// TIA Portal V15.1 export
// export: Created 2020-12-07T09:03:51.8959299Z, ExportSetting WithDefaults, WithReadOnly, DisplayName Totally Integrated Automation Portal, DisplayVersion V15.1 Update 4, DisplayName TIA Portal Openness, DisplayVersion V15.1, DisplayName SINAMICS Startdrive Advanced, DisplayVersion V15.1 Update3, DisplayName SINAMICS Startdrive G110M, G120, G120C, G120D, G120P, DisplayVersion V15.1 Update3, DisplayName SINAMICS Startdrive G130, G150, S120, S150, SINAMICS MV, S210, DisplayVersion V15.1 Update3, DisplayName STEP 7 Professional, DisplayVersion V15.1 Update 4, DisplayName STEP 7 Safety, DisplayVersion V15.1, DisplayName WinCC Professional, DisplayVersion V15.1 Update 4
VAR_GLOBAL   // PLC tag table "INPUT_ST_A"
   "SQ84/BA" AT %I2000.0 : Bool;
   "SQ85/BA" AT %I2001.0 : Bool;
   "SQ86/BA" AT %I2000.1 : Bool;
   "SQ87/BA" AT %I2001.1 : Bool;
   "SQ57/BA" AT %I2000.2 : Bool;
   "SQ58/BA" AT %I2001.2 : Bool;
   "SQ59/BA" AT %I2000.3 : Bool;
   "SQ60/BA" AT %I2001.3 : Bool;
   "SQ73/BA" AT %I2000.4 : Bool;
   "SQ74/BA" AT %I2001.4 : Bool;
   "SQ31/BA" AT %I2000.5 : Bool;
   "SQ32/BA" AT %I2001.5 : Bool;
   "FTC1/BA" AT %I2000.7 : Bool;
   "SQ15/BA" AT %I2001.6 : Bool;
   "FTC2/BA" AT %I2000.6 : Bool;
   "FTC3/BA" AT %I2001.7 : Bool;
   "SQ61/BA" AT %I2002.0 : Bool;
   "SQ62/BA" AT %I2003.0 : Bool;
   "SQ66/BA" AT %I2002.1 : Bool;
   "SQ67/BA" AT %I2003.1 : Bool;
   "SQ68/BA" AT %I2002.2 : Bool;
   "SQ72/BA" AT %I2003.2 : Bool;
   "SQ8/BA" AT %I2002.3 : Bool;   // // NC
   "SQ9/BA" AT %I2003.3 : Bool;   // // NC
   "SQ80/BA" AT %I2002.4 : Bool;
   "SQ81/BA" AT %I2003.4 : Bool;
   "FTC15/BA" AT %I2002.5 : Bool;   // Scivolo troppo pieno
   "FTC92/BA" AT %I2003.5 : Bool;   // Presenza rullo su OP30
   "FTC93/BA" AT %I2002.6 : Bool;   // Presenza rullo su OP20
   "FTC94/BA" AT %I2003.6 : Bool;   // Presenza rullo su OP10
   "SQ_SPARE_31/BA" AT %I2002.7 : Bool;
   "SQ_SPARE_32/BA" AT %I2003.7 : Bool;
   "SQ_SPARE_33/BA" AT %I2004.0 : Bool;   // // NC
   "SQ_SPARE_34/BA" AT %I2005.0 : Bool;   // // NC
   "SQ_SPARE_35/BA" AT %I2004.1 : Bool;   // // NC
   "SQ_SPARE_36/BA" AT %I2005.1 : Bool;   // // NC
   "SQ_SPARE_37/BA" AT %I2004.2 : Bool;   // // NC
   "SQ_SPARE_38/BA" AT %I2005.2 : Bool;   // // NC
   "SQ_SPARE_39/BA" AT %I2004.3 : Bool;
   "SQ_SPARE_40/BA" AT %I2005.3 : Bool;
   "SQ_SPARE_41/BA" AT %I2004.4 : Bool;
   "SQ_SPARE_42/BA" AT %I2005.4 : Bool;
   "SQ_SPARE_43/BA" AT %I2004.5 : Bool;
   "SQ_SPARE_44/BA" AT %I2005.5 : Bool;
   "SQ_SPARE_45/BA" AT %I2004.6 : Bool;
   "SQ_SPARE_46/BA" AT %I2005.6 : Bool;
   "SQ_SPARE_47/BA" AT %I2004.7 : Bool;
   "SQ_SPARE_48/BA" AT %I2005.7 : Bool;
   "SQ44/BA" AT %I2100.0 : Bool;
   "SQ45/BA" AT %I2101.0 : Bool;
   "SQ88/BA" AT %I2100.1 : Bool;
   "SQ89/BA" AT %I2101.1 : Bool;
   "SQ48/BA" AT %I2100.2 : Bool;
   "SQ49/BA" AT %I2101.2 : Bool;
   "SQ50/BA" AT %I2100.3 : Bool;
   "SQ51/BA" AT %I2101.3 : Bool;
   "SQ75/BA" AT %I2100.4 : Bool;
   "SQ76/BA" AT %I2101.4 : Bool;
   "SQ18/BA" AT %I2100.5 : Bool;
   "SQ19/BA" AT %I2101.5 : Bool;
   "SQ97/BA" AT %I2100.6 : Bool;
   "SQ17/BA" AT %I2101.6 : Bool;
   "SQ98/BA" AT %I2100.7 : Bool;
   "SQ_SPARE_64/BA" AT %I2101.7 : Bool;
   "SQ_SPARE_65/BA" AT %I2102.0 : Bool;   // // NC
   "SQ_SPARE_66/BA" AT %I2103.0 : Bool;   // // NC
   "SQ_SPARE_67/BA" AT %I2102.1 : Bool;   // // NC
   "SQ_SPARE_68/BA" AT %I2103.1 : Bool;   // // NC
   "SQ_SPARE_69/BA" AT %I2102.2 : Bool;   // // NC
   "SQ_SPARE_70/BA" AT %I2103.2 : Bool;   // // NC
   "SQ_SPARE_71/BA" AT %I2102.3 : Bool;
   "SQ_SPARE_72/BA" AT %I2103.3 : Bool;
   "SQ_SPARE_73/BA" AT %I2102.4 : Bool;
   "SQ_SPARE_74/BA" AT %I2103.4 : Bool;
   "SQ_SPARE_75/BA" AT %I2102.5 : Bool;
   "SQ_SPARE_76/BA" AT %I2103.5 : Bool;
   "SQ_SPARE_77/BA" AT %I2102.6 : Bool;
   "SQ_SPARE_78/BA" AT %I2103.6 : Bool;
   "SQ_SPARE_79/BA" AT %I2102.7 : Bool;
   "SQ_SPARE_80/BA" AT %I2103.7 : Bool;
   "SQ69/BA" AT %I2104.0 : Bool;
   "SQ70/BA" AT %I2105.0 : Bool;
   "SQ71/BA" AT %I2104.1 : Bool;
   "SQ77/BA" AT %I2105.1 : Bool;
   "SQ78/BA" AT %I2104.2 : Bool;
   "SQ79/BA" AT %I2105.2 : Bool;   // // NC
   "SQ6/BA" AT %I2104.3 : Bool;
   "SQ7/BA" AT %I2105.3 : Bool;
   "SQ82/BA" AT %I2104.4 : Bool;
   "SQ83/BA" AT %I2105.4 : Bool;
   "SQ_SPARE_91/BA" AT %I2104.5 : Bool;
   "SQ_SPARE_92/BA" AT %I2105.5 : Bool;
   "SQ_SPARE_93/BA" AT %I2104.6 : Bool;
   "SQ_SPARE_94/BA" AT %I2105.6 : Bool;
   "SQ_SPARE_95/BA" AT %I2104.7 : Bool;
   "SQ_SPARE_96/BA" AT %I2105.7 : Bool;
   "STO_AZ2/BA" AT %I4.0 : Bool;   // // NC
   "STO_AZ3/BA" AT %I4.1 : Bool;   // // NC
   "STO_AZ11/BA" AT %I4.2 : Bool;   // // NC
   "STO_AZ14/BA" AT %I4.3 : Bool;   // // NC
   "STO_AZ18/BA" AT %I4.4 : Bool;   // // NC
   "STO_AZ20/BA" AT %I4.5 : Bool;   // // NC
   "STO_AZ22/BA" AT %I4.6 : Bool;   // // NC
   "STO_AZ24/BA" AT %I4.7 : Bool;   // // NC
   "STO_AZ4/BA" AT %I5.0 : Bool;   // // NC
   "STO_AZ5/BA" AT %I5.1 : Bool;   // // NC
   "STO_AZ6/BA" AT %I5.2 : Bool;   // // NC
   "STO_AZ7/BA" AT %I5.3 : Bool;   // // NC
   "STO_AZ8/BA" AT %I5.4 : Bool;   // // NC
   "STO_AZ9/BA" AT %I5.5 : Bool;   // // NC
   "STO_AZ10/BA" AT %I5.6 : Bool;   // // NC
   "STO_AZ12/BA" AT %I5.7 : Bool;   // // NC
   "STO_AZ13/BA" AT %I6.0 : Bool;   // // NC
   "STO_AZ15/BA" AT %I6.1 : Bool;   // // NC
   "STO_AZ17/BA" AT %I6.2 : Bool;   // // NC
   "STO_AZ19/BA" AT %I6.3 : Bool;   // // NC
   "STO_AZ21/BA" AT %I6.4 : Bool;   // // NC
   "STO_AZ23/BA" AT %I6.5 : Bool;   // // NC
   "STO_AZ25/BA" AT %I6.6 : Bool;   // // NC
   "STO_AZ26/BA" AT %I6.7 : Bool;   // // NC
   "OIL_PUMP_FAULT/BA" AT %I7.0 : Bool;
   "EMG_OK/BA" AT %I7.1 : Bool;
   "OIL_HIGH_TEMP/BA" AT %I7.2 : Bool;
   "OIL_LOW_LEVEL/BA" AT %I7.3 : Bool;
   "LASER_ERROR/BA" AT %I7.4 : Bool;   // // NC
   "AZ27_RUN/BA" AT %I7.6 : Bool;   // // NC
   "AZ27_FAULT/BA" AT %I7.7 : Bool;   // // NC
   "LOAD_CELL_SX_FAULT/BA" AT %I8.0 : Bool;
   "PS_KOSTYRCA_ENDCAP_SX/BA" AT %I8.1 : Bool;
   "PS_KOSTYRCA_SEEGER_SX/BA" AT %I8.2 : Bool;
   "PS_KOSTYRCA_ENDCAP_DX/BA" AT %I8.3 : Bool;
   "PS_KOSTYRCA_SEEGER_DX/BA" AT %I8.4 : Bool;
   "LOAD_CELL_DX_FAULT/BA" AT %I8.5 : Bool;
   "TLB1/BA" AT %IW2 : Int;   // Load cell endcap sx
   "TLB2/BA" AT %IW0 : Int;   // Load cell endcap dx
   "TOR1/BA" AT %IW10 : Int;   // Torsiometro
   "FTC5/BA" AT %I2006.0 : Bool;
   "FTC7/BA" AT %I2006.1 : Bool;
   "SQ_SPARE_99/BA" AT %I2006.2 : Bool;
   "FTC90/BA" AT %I2006.3 : Bool;   // Presenza Endcap SX
   "SQ_SPARE_101/BA" AT %I2006.4 : Bool;
   "SQ_SPARE_102/BA" AT %I2006.5 : Bool;
   "SQ_SPARE_103/BA" AT %I2006.6 : Bool;
   "SQ_SPARE_104/BA" AT %I2006.7 : Bool;
   "FTC6/BA" AT %I2007.0 : Bool;
   "SQ95/BA" AT %I2007.1 : Bool;
   "SQ_SPARE_107/BA" AT %I2007.2 : Bool;
   "SQ96/BA" AT %I2007.3 : Bool;
   "SQ_SPARE_109/BA" AT %I2007.4 : Bool;
   "SQ_SPARE_110/BA" AT %I2007.5 : Bool;
   "SQ_SPARE_111/BA" AT %I2007.6 : Bool;
   "SQ_SPARE_112/BA" AT %I2007.7 : Bool;
   "SQ_SPARE_113/BA" AT %I2106.0 : Bool;
   "SQ_SPARE_114/BA" AT %I2106.1 : Bool;
   "SQ_SPARE_115/BA" AT %I2106.2 : Bool;
   "SQ_SPARE_116/BA" AT %I2106.3 : Bool;
   "FTC91/BA" AT %I2106.4 : Bool;   // Presenza Endcap DX
   "SQ_SPARE_118/BA" AT %I2106.5 : Bool;
   "SQ_SPARE_119/BA" AT %I2106.6 : Bool;
   "SQ_SPARE_120/BA" AT %I2106.7 : Bool;
   "SQ_SPARE_121/BA" AT %I2107.0 : Bool;
   "SQ_SPARE_122/BA" AT %I2107.1 : Bool;
   "SQ_SPARE_123/BA" AT %I2107.2 : Bool;
   "SQ_SPARE_124/BA" AT %I2107.3 : Bool;
   "SQ_SPARE_125/BA" AT %I2107.4 : Bool;
   "SQ_SPARE_126/BA" AT %I2107.5 : Bool;
   "SQ_SPARE_127/BA" AT %I2107.6 : Bool;
   "SQ_SPARE_128/BA" AT %I2107.7 : Bool;
   "Raw_KEYENCE_IL10xx_LS1/BA" AT %ID2353 : DInt;
   "Raw_KEYENCE_IL10xx_LS2/BA" AT %ID2363 : DInt;
   "Raw_KEYENCE_IL10xx_LS3/BA" AT %ID2373 : DInt;
   "OIL_IN_PRESSURE/BA" AT %I8.6 : Bool;   // // NC
END_VAR
